// SIMATIC S7-200 SMART project (STEP 7-Micro/WIN SMART), CPU SR40

ORGANIZATION_BLOCK 主程序:OB1
TITLE=程序注释
BEGIN
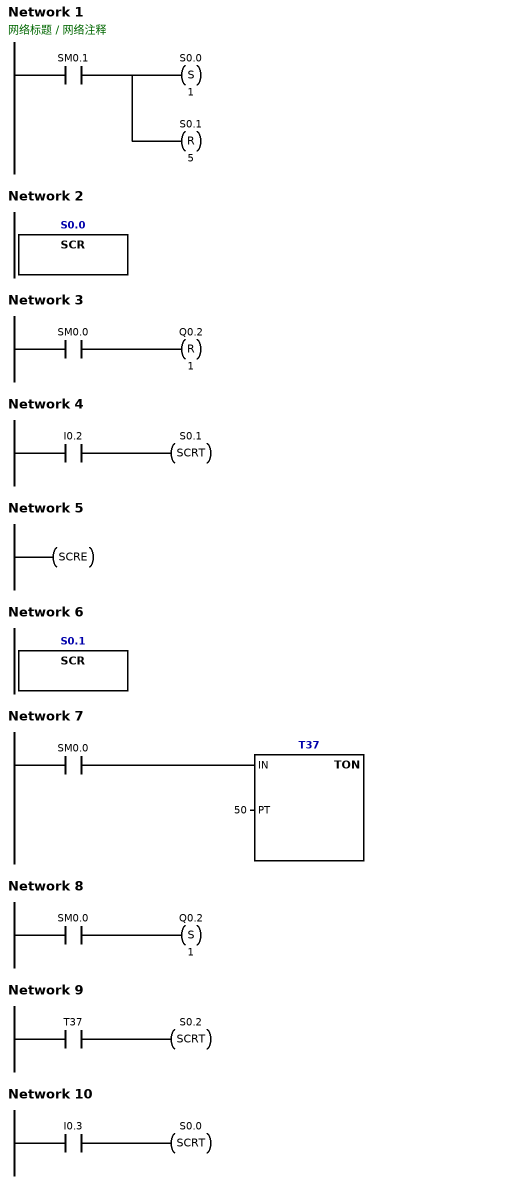
Network 1
// 网络标题
// 网络注释
LD     SM0.1
S      S0.0, 1
R      S0.1, 5
Network 2
LSCR   S0.0
Network 3
LD     SM0.0
R      Q0.2, 1
Network 4
LD     I0.2
SCRT   S0.1
Network 5
SCRE
Network 6
LSCR   S0.1
Network 7
// (network saved uncompiled; LAD cells follow)
// row 0: c0 -| |- SM0.0  c1 --  c2 [TON T37 IN:=power@row0, PT:=50]
// row 1: c2 [box]
Network 8
LD     SM0.0
S      Q0.2, 1
Network 9
LD     T37
SCRT   S0.2
Network 10
LD     I0.3
SCRT   S0.0
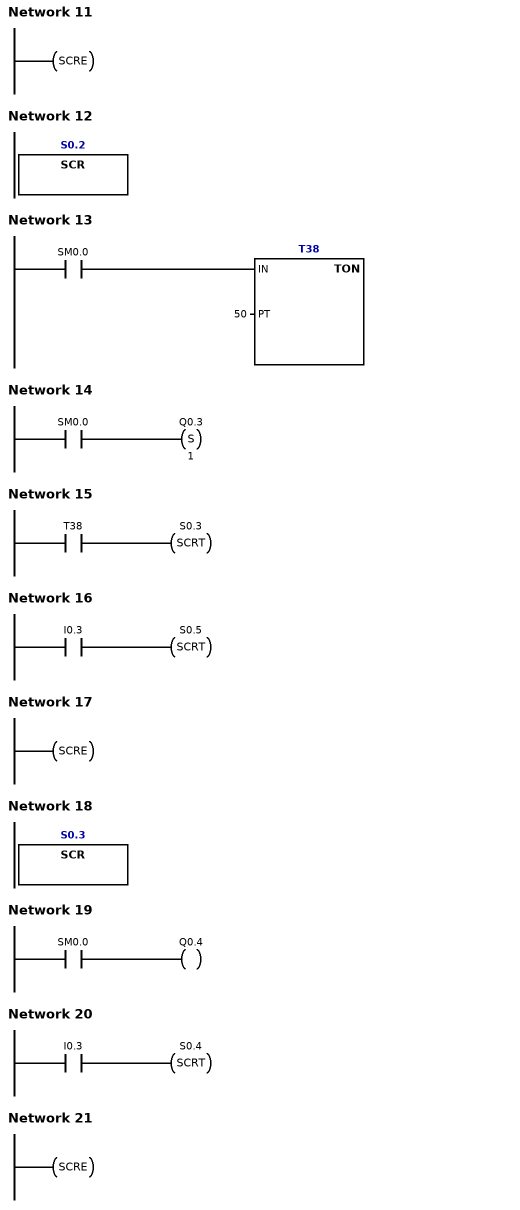
Network 11
SCRE
Network 12
LSCR   S0.2
Network 13
// (network saved uncompiled; LAD cells follow)
// row 0: c0 -| |- SM0.0  c1 --  c2 [TON T38 IN:=power@row0, PT:=50]
// row 1: c2 [box]
Network 14
LD     SM0.0
S      Q0.3, 1
Network 15
LD     T38
SCRT   S0.3
Network 16
LD     I0.3
SCRT   S0.5
Network 17
SCRE
Network 18
LSCR   S0.3
Network 19
LD     SM0.0
=      Q0.4
Network 20
LD     I0.3
SCRT   S0.4
Network 21
SCRE
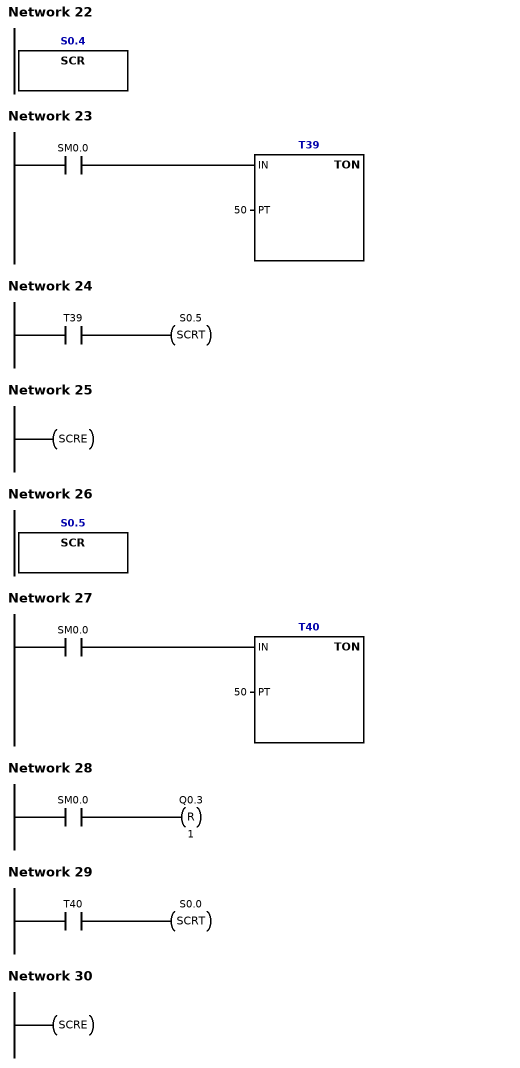
Network 22
LSCR   S0.4
Network 23
// (network saved uncompiled; LAD cells follow)
// row 0: c0 -| |- SM0.0  c1 --  c2 [TON T39 IN:=power@row0, PT:=50]
// row 1: c2 [box]
Network 24
LD     T39
SCRT   S0.5
Network 25
SCRE
Network 26
LSCR   S0.5
Network 27
// (network saved uncompiled; LAD cells follow)
// row 0: c0 -| |- SM0.0  c1 --  c2 [TON T40 IN:=power@row0, PT:=50]
// row 1: c2 [box]
Network 28
LD     SM0.0
R      Q0.3, 1
Network 29
LD     T40
SCRT   S0.0
Network 30
SCRE
END_ORGANIZATION_BLOCK
